# EPICS StreamDevice protocol: nomad-camels/instruments/agilent_34401/camels_driver_agilent_34401/agilent_34401.proto
ReplyTimeout = 2000;
InTerminator = CR LF;

#Measure voltage DC
mesDCV {
	out "MEAS:VOLT:DC?";
	in "%f";
    ExtraInput = Ignore;
}

#Measure current DC
mesDCI {
	out "MEAS:CURR:DC?";
	in "%f";
    ExtraInput = Ignore;
}

#Measure voltage AC
mesACV {
	out "MEAS:VOLT:AC?";
	in "%f";
    ExtraInput = Ignore;
}

#Measure current AC
mesACI {
	out "MEAS:CURR:AC?";
	in "%f";
    ExtraInput = Ignore;
}

#Measure Resistance
#2 wire
mesR {
	out "MEAS:RES?";
	in "%f";
    ExtraInput = Ignore;
}

#4 wire
mesR4 {
	out "MEAS:FRES?";
	in "%f";
	ExtraInput = Ignore;
}

#nPLC, integration time
nPLC {
	out "VOLT:DC:NPLC %f";
	out "VOLT:AC:NPLC %f";
	out "CURR:DC:NPLC %f";
	out "CURR:AC:NPLC %f";
	out "RES:NPLC %f";
	out "FRES:NPLC %f";
}

#get Identification

idn {
	out "*IDN?";
	in "%[^\r\n]";
    ExtraInput = Ignore;
}
